PROGRAM StartUpTests
VAR CONSTANT
	stPlcErrorInit			: ST_PlcErrorStartUp := (bPlcError := FALSE, bErrorCode := [0,0,0,0]);
END_VAR

VAR
	eStartUpState 			: (WAIT_FOR_TRIGGER, TEST_SWITCH_ON_DISABLED, 
								SET_MODE_OF_OPERATION, TEST_MODE_OF_OPERATION, GET_TEMPERATURE, CHECK_PLC_ERROR);
	fbSetModeOfOperation	: FB_EcCoeSdoWrite;
	fbGetModeOfOperation	: FB_EcCoeSdoRead;
	fbGetDriveTemperature	: FB_EcCoeSdoRead;
	fbGetMotorTemperature	: FB_EcCoeSdoRead;
	stPlcError				: ST_PlcErrorStartUp;
	tTimeout				: TON;
	tWait1					: TON;
	tWait2					: TON;
	tWait					: TON;
	counter					: INT := -1;
	modeOfOperation			: INT;
	bExecuteChangeMOP		: BOOL;	
	bTestChangeMOP			: BOOL;
END_VAR
VAR_IN_OUT
	bTrigger				: BOOL;
	aTemperatureObjects		: ARRAY[1..2] OF INT;
	aMOPObjects				: ARRAY[1..2] OF INT;
	aControlStatusWords		: ARRAY[1..2] OF INT;
END_VAR
VAR_OUTPUT
	bSwitchOnDisabled		: BOOL;
	bChangeModeOfOperation	: BOOL := TRUE;
	bFinished				: BOOL;
	nDriveTemperature		: INT;
	nMotorTemperature		: INT;
END_VAR
VAR_INPUT
	sNetID					: T_AmsNetId;
	nSlaveAddr				: UINT;
END_VAR

CASE eStartUpState OF
	WAIT_FOR_TRIGGER:
		IF bTrigger THEN
			bTrigger := FALSE;
			tTimeout.IN := FALSE;
			bSwitchOnDisabled := FALSE;
			bChangeModeOfOperation := FALSE;
			bFinished := FALSE;
			counter := 1;
			stPlcError := stPlcErrorInit;
			eStartUpState := TEST_SWITCH_ON_DISABLED;
		END_IF
	
	TEST_SWITCH_ON_DISABLED:
		tTimeout(IN := TRUE,
			PT := T#1000MS);
		IF MAIN.Statusword.6 THEN
			bSwitchOnDisabled := TRUE;
			eStartUpState := SET_MODE_OF_OPERATION;
		ELSIF tTimeout.Q THEN
			bSwitchOnDisabled := FALSE;
			aControlStatusWords[1] := 0;
			eStartUpState := SET_MODE_OF_OPERATION;
		END_IF
	
	SET_MODE_OF_OPERATION:
	bTestChangeMOP := FALSE;
		fbSetModeOfOperation(sNetId := sNetId,
							nSlaveAddr := nSlaveAddr,
							nSubIndex := 0,
							nIndex := 16#6060,
							pSrcBuf := ADR(counter),
							cbBufLen := SIZEOF(counter),
							bExecute := bExecuteChangeMOP);
		tWait1(PT := T#2S, 
			IN := bExecuteChangeMOP);
		bExecuteChangeMOP := TRUE;				
		IF tWait1.Q THEN
			eStartUpState := TEST_MODE_OF_OPERATION;
		END_IF

	TEST_MODE_OF_OPERATION:
		bExecuteChangeMOP := FALSE;	
		fbGetModeOfOperation(sNetId := sNetId,
							nSlaveAddr := nSlaveAddr,
							nSubIndex := 0,
							nIndex := 16#6061,
							pDstBuf := ADR(modeOfOperation),
							cbBufLen := SIZEOF(modeOfOperation),
							bExecute := bTestChangeMOP);
		tWait2(PT := T#2S,
				IN := bTestChangeMOP);
		bTestChangeMOP := TRUE; 
		IF tWait2.Q THEN
			IF NOT modeOfOperation = counter AND counter <> 5 THEN
				bChangeModeOfOperation := FALSE;
				aMOPObjects[1] := 0;
				aMOPObjects[2] := 0;
			END_IF
			counter := counter + 1;
			IF counter < 11 THEN
				eStartUpState := SET_MODE_OF_OPERATION;
			ELSE
				eStartUpState := GET_TEMPERATURE;
			END_IF
		END_IF
	
	GET_TEMPERATURE:
		fbGetDriveTemperature(sNetId := sNetId,
							nSlaveAddr := nSlaveAddr,
							nSubIndex := 0,
							nIndex := 16#2200,
							pDstBuf := ADR(nDriveTemperature),
							cbBufLen := SIZEOF(nDriveTemperature),
							bExecute := TRUE);
		fbGetMotorTemperature(sNetId := sNetId,
							nSlaveAddr := nSlaveAddr,
							nSubIndex := 0,
							nIndex := 16#2202,
							pDstBuf := ADR(nMotorTemperature),
							bExecute := TRUE);							
		tWait(IN := TRUE,
			PT := T#125MS);
		IF tWait.Q THEN
			tWait.IN := FALSE;
		//	eStartUpState := CHECK_PLC_ERROR;
		END_IF
		
		CHECK_PLC_ERROR:
			IF fbSetModeOfOperation.bError OR fbGetModeOfOperation.bError OR
				fbGetDriveTemperature.bError OR fbGetMotorTemperature.bError THEN
				stPlcError.bPlcError := TRUE;
				IF fbSetModeOfOperation.bError THEN
					stPlcError.bErrorCode[1] := fbSetModeOfOperation.nErrId;
					aMOPObjects[1] := 0;
				END_IF
				IF fbGetModeOfOperation.bError THEN
					stPlcError.bErrorCode[2] := fbGetModeOfOperation.nErrId;
					aMOPObjects[2] := 0;		
				END_IF
				IF fbGetDriveTemperature.bError THEN
					stPlcError.bErrorCode[3] := fbGetDriveTemperature.nErrId;
					aTemperatureObjects[1] := 0;
				END_IF
				IF fbGetMotorTemperature.bError THEN
					stPlcError.bErrorCode[4] := fbGetMotorTemperature.nErrId;
					aTemperatureObjects[2] := 0;
				END_IF
			END_IF
			bFinished := TRUE;
			eStartUpState := WAIT_FOR_TRIGGER;
END_CASE

END_PROGRAM

(* stored: Version 1.1.0.1, ProductVersion 3.1.4024.11
   POU StartUpTests: Id {5c2c3321-b140-4518-a103-c3096216c8a3}, SpecialFunc None *)
